GLOBALCONSTANTS IG4_Device_Classes (* Industry Group 4 specific device classes (vehicle systems) *)
  (* Standard: 61499-1 *)
  (* Version 1.0, 2026-06-30, Franz Höpfinger, Demmler Andreas Fahrzeugbau *)
  PACKAGE isobus::pgn::const;
  VAR_GLOBAL CONSTANT
    DC_NON_SPECIFIC_SYSTEM : BYTE := 0; (* Device Class / Vehicle System: Non-specific System *)
    DC_SYSTEM_TOOLS : BYTE := 10; (* Device Class / Vehicle System: System tools *)
    DC_SAFETY_SYSTEMS : BYTE := 20; (* Device Class / Vehicle System: Safety systems *)
    DC_GATEWAY : BYTE := 25; (* Device Class / Vehicle System: Gateway *)
    DC_POWER_MGMT_LIGHTING : BYTE := 30; (* Device Class / Vehicle System: Power management and lighting systems *)
    DC_STEERING_SYSTEMS : BYTE := 40; (* Device Class / Vehicle System: Steering systems *)
    DC_PROPULSION_SYSTEMS : BYTE := 50; (* Device Class / Vehicle System: Propulsion systems *)
    DC_NAVIGATION_SYSTEMS : BYTE := 60; (* Device Class / Vehicle System: Navigation systems *)
    DC_COMMUNICATIONS_SYSTEMS : BYTE := 70; (* Device Class / Vehicle System: Communications systems *)
    DC_INSTRUMENTATION_GENERAL : BYTE := 80; (* Device Class / Vehicle System: Instrumentation/general systems *)
    DC_ENVIRONMENTAL_HVAC : BYTE := 90; (* Device Class / Vehicle System: Environmental (HVAC) systems *)
    DC_DECK_CARGO_FISHING : BYTE := 100; (* Device Class / Vehicle System: Deck, cargo, and fishing equipment systems *)
    DC_NOT_AVAILABLE : BYTE := 127; (* Device Class / Vehicle System: Not Available *)
  END_VAR
END_GLOBALCONSTANTS
